{attribute addProperty BoxType "AX8108-0000-0041-0041"}
{attribute addProperty Id "DeviceMain_OutputsDeviceMain_Outputs_04240708162"}
{attribute addProperty CRC "4249400496"}
{attribute addProperty SizeInBites "16"}
{attribute addProperty SizeInBytes "2"}
TYPE Device_FD48B4B0 :
STRUCT
	{attribute addProperty Name "DeviceMain_Outputs"}
	DeviceMain_Outputs  : DeviceMain_Outputs_04240708;
END_STRUCT
END_TYPE

(* stored: Version 1.2.0.0, ProductVersion 3.1.4024.9
   DUT Device_FD48B4B0: Id {6426763b-5022-4cca-a564-d51295c94324} *)
